PROGRAM Alarm_Logic
VAR
	
	RedStack		:	Blink;
	YellowStack		:	Blink;
	BlueStack		:	Blink;
	YellowLED		:	Blink;
	
END_VAR


IF Pump.LLSwicth AND Pump.HHSwitch = FALSE THEN

	RedStack(Enable := TRUE, Period := T#125MS ,Q=> Pump.RedLED);
	YellowStack(Enable := TRUE, Period := T#125MS ,Q=> Pump.YellowLED);	

END_IF

END_PROGRAM

(* stored: Version 1.1.0.1, ProductVersion 3.1.4024.9
   POU Alarm_Logic: Id {4c516ebb-c9a1-4afb-b6ad-18be282a697b}, SpecialFunc None *)
